{attribute 'qualified_only'}
VAR_GLOBAL
	m_curLinkPos :ARRAY[1..2] OF Vec7d;
	m_curJntPos :ARRAY[1..2] OF Vec7d;
	m_JntGap :ARRAY[1..2] OF Vec7d;
END_VAR

(* stored: Version 1.1.0.1, ProductVersion 3.1.4024.11
   GVL GVL: Id {312f603e-a9dd-4715-8ff2-a916db41d175} *)
